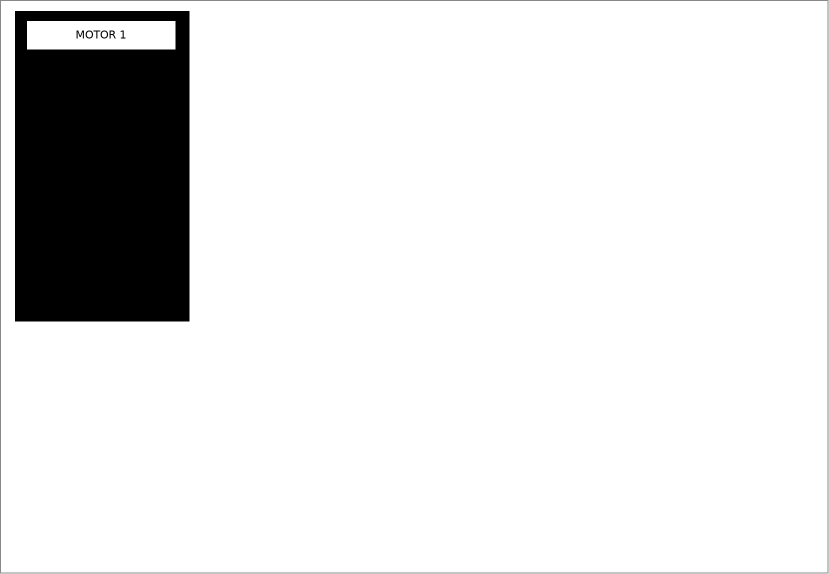
VISUALIZATION machineMapScreen  // 829x574
    Rectangle (15,11 174x310)
    Rectangle (26,20 150x30), "MOTOR 1"
END_VISUALIZATION

(* stored: Version 1.1.0.1, ProductVersion 3.1.4024.15
   Visu machineMapScreen: Id {38e19128-55c1-4aa5-9ab6-0d4856cb7fe6} *)
